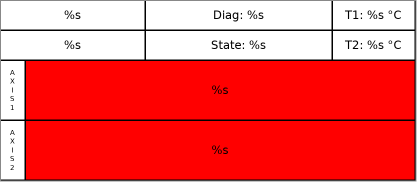
VISUALIZATION TplTsConnectionAX5805  // 417x182
VAR_IN_OUT
	stConnectionDiag 			:FB_TwinSafeConnectionAX5805;
END_VAR
(* End *)
    Rectangle (0,0 145x30), "%s", text variable: stConnectionDiag.sEcSlaveName
    Rectangle (25,60 49x30), "S-STO", colour toggle: stConnectionDiag.stSignalStatusMC1.bSafeTorqueOff_STO
    Rectangle (74,60 49x30), "S-SMM1", colour toggle: stConnectionDiag.stSignalStatusMC1.bSafeSpeedMonitor_SSM_1
    Rectangle (123,60 49x30), "S-SSM2", colour toggle: stConnectionDiag.stSignalStatusMC1.bSafeSpeedMonitor_SSM_2
    Rectangle (172,60 48x30), "S-SOS1", colour toggle: stConnectionDiag.stSignalStatusMC1.bSafeOperatingStop_SOS_1
    Rectangle (145,0 187x30), "Diag: %s", text variable: stConnectionDiag.sDiag, colour toggle: stConnectionDiag.sDiag <> 'No error'
    Rectangle (145,30 187x30), "State: %s", text variable: stConnectionDiag.sState
    Rectangle (0,30 145x30), "%s", text variable: stConnectionDiag.sEcSlaveType
    Rectangle (220,60 49x30), "S-SSR1", colour toggle: stConnectionDiag.stSignalStatusMC1.bSafeSpeedRange_SSR_1
    Rectangle (269,60 49x30), "S-SDIp", colour toggle: stConnectionDiag.stSignalStatusMC1.bSafeDirectionPositive_SDIp
    Rectangle (318,60 49x30), "S-SDIn", colour toggle: stConnectionDiag.stSignalStatusMC1.bSafeDirectionNegative_SDIn
    Rectangle (367,60 48x30), "S-Err Ack", colour toggle: stConnectionDiag.stSignalStatusMC1.bErrorAcknowledge_ErrAck
    Rectangle (25,90 49x30), "C-STO", colour toggle: stConnectionDiag.stSignalControlStatusMC1.bSafeTorqueOff_STO
    Rectangle (74,90 49x30), "C-SS1", colour toggle: stConnectionDiag.stSignalControlStatusMC1.bSafeStop1_SS1_1
    Rectangle (123,90 49x30), "C-SS2", colour toggle: stConnectionDiag.stSignalControlStatusMC1.bSafeStop2_SS2_1
    Rectangle (172,90 48x30), "C-SOS1", colour toggle: stConnectionDiag.stSignalControlStatusMC1.bSafeOperatingStop_SOS_1
    Rectangle (220,90 49x30), "C-SSR1", colour toggle: stConnectionDiag.stSignalControlStatusMC1.bSafeSpeedRange_SSR_1
    Rectangle (269,90 49x30), "C-SDIp", colour toggle: stConnectionDiag.stSignalControlStatusMC1.bSafeDirectionPositive_SDIp
    Rectangle (318,90 49x30), "C-SDIn", colour toggle: stConnectionDiag.stSignalControlStatusMC1.bSafeDirectionNegative_SDIn
    Rectangle (367,90 48x30), "C-Err Ack", colour toggle: stConnectionDiag.stSignalControlStatusMC1.bErrorAcknowledge_ErrAck
    Rectangle (332,0 83x30), "T1: %s °C", text variable: stConnectionDiag.stSlaveTemp.nInternalTemperature1, colour toggle: stConnectionDiag.bTempWarning
    Rectangle (332,30 83x30), "T2: %s °C", text variable: stConnectionDiag.stSlaveTemp.nInternalTemperature2, colour toggle: stConnectionDiag.bTempWarning
    Rectangle (25,120 49x30), "S-STO", colour toggle: stConnectionDiag.stSignalStatusMC2.bSafeTorqueOff_STO
    Rectangle (74,120 49x30), "S-SMM1", colour toggle: stConnectionDiag.stSignalStatusMC2.bSafeSpeedMonitor_SSM_1
    Rectangle (123,120 49x30), "S-SSM2", colour toggle: stConnectionDiag.stSignalStatusMC2.bSafeSpeedMonitor_SSM_2
    Rectangle (172,120 48x30), "S-SOS1", colour toggle: stConnectionDiag.stSignalStatusMC2.bSafeOperatingStop_SOS_1
    Rectangle (220,120 49x30), "S-SSR1", colour toggle: stConnectionDiag.stSignalStatusMC2.bSafeSpeedRange_SSR_1
    Rectangle (269,120 49x30), "S-SDIp", colour toggle: stConnectionDiag.stSignalStatusMC2.bSafeDirectionPositive_SDIp
    Rectangle (318,120 49x30), "S-SDIn", colour toggle: stConnectionDiag.stSignalStatusMC2.bSafeDirectionNegative_SDIn
    Rectangle (367,120 48x30), "S-Err Ack", colour toggle: stConnectionDiag.stSignalStatusMC2.bErrorAcknowledge_ErrAck
    Rectangle (25,150 49x30), "C-STO", colour toggle: stConnectionDiag.stSignalControlStatusMC2.bSafeTorqueOff_STO
    Rectangle (74,150 49x30), "C-SS1", colour toggle: stConnectionDiag.stSignalControlStatusMC2.bSafeStop1_SS1_1
    Rectangle (123,150 49x30), "C-SS2", colour toggle: stConnectionDiag.stSignalControlStatusMC2.bSafeStop2_SS2_1
    Rectangle (172,150 48x30), "C-SOS1", colour toggle: stConnectionDiag.stSignalControlStatusMC2.bSafeOperatingStop_SOS_1
    Rectangle (220,150 49x30), "C-SSR1", colour toggle: stConnectionDiag.stSignalControlStatusMC2.bSafeSpeedRange_SSR_1
    Rectangle (269,150 49x30), "C-SDIp", colour toggle: stConnectionDiag.stSignalControlStatusMC2.bSafeDirectionPositive_SDIp
    Rectangle (318,150 49x30), "C-SDIn", colour toggle: stConnectionDiag.stSignalControlStatusMC2.bSafeDirectionNegative_SDIn
    Rectangle (367,150 48x30), "C-Err Ack", colour toggle: stConnectionDiag.stSignalControlStatusMC2.bErrorAcknowledge_ErrAck
    Rectangle (0,60 25x60), "A X I S 1"
    Rectangle (0,120 25x60), "A X I S 2"
    Rectangle (26,61 388x58), "%s", text variable: stConnectionDiag.eErrIndicesFA82DiagnosisMC1, invisible if: NOT stConnectionDiag.bErrIndicesFA82DiagnosisMC1Err
    Rectangle (26,121 388x58), "%s", text variable: stConnectionDiag.eErrIndicesFA82DiagnosisMC2, invisible if: NOT stConnectionDiag.bErrIndicesFA82DiagnosisMC2Err
END_VISUALIZATION

(* stored: Version 1.1.0.1
   Visu TplTsConnectionAX5805: Id {ebc13c06-03a0-468f-97b1-e8a49526fd41} *)
